FUNCTION_BLOCK Valvula_Saida_Digital (* Composite Function Block Type *)
  (* Standard: 61499-2 *)
  (* Version 0.0, 1/26/2026, Schneider Electric, template *)
  PACKAGE Hidryco.HidrycoLib;
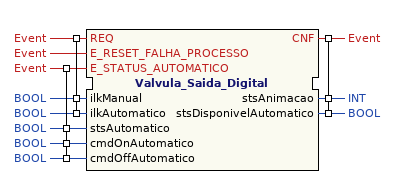
  EVENT_INPUT
    REQ WITH ilkManual, ilkAutomatico; (* Normal Execution Request *)
    E_RESET_FALHA_PROCESSO;
    E_STATUS_AUTOMATICO WITH cmdOnAutomatico, cmdOffAutomatico, stsAutomatico;
  END_EVENT
  EVENT_OUTPUT
    CNF WITH stsAnimacao, stsDisponivelAutomatico;
  END_EVENT
  VAR_INPUT
    ilkManual : BOOL;
    ilkAutomatico : BOOL;
    stsAutomatico : BOOL;
    cmdOnAutomatico : BOOL;
    cmdOffAutomatico : BOOL;
  END_VAR
  VAR_OUTPUT
    stsAnimacao : INT;
    stsDisponivelAutomatico : BOOL;
  END_VAR
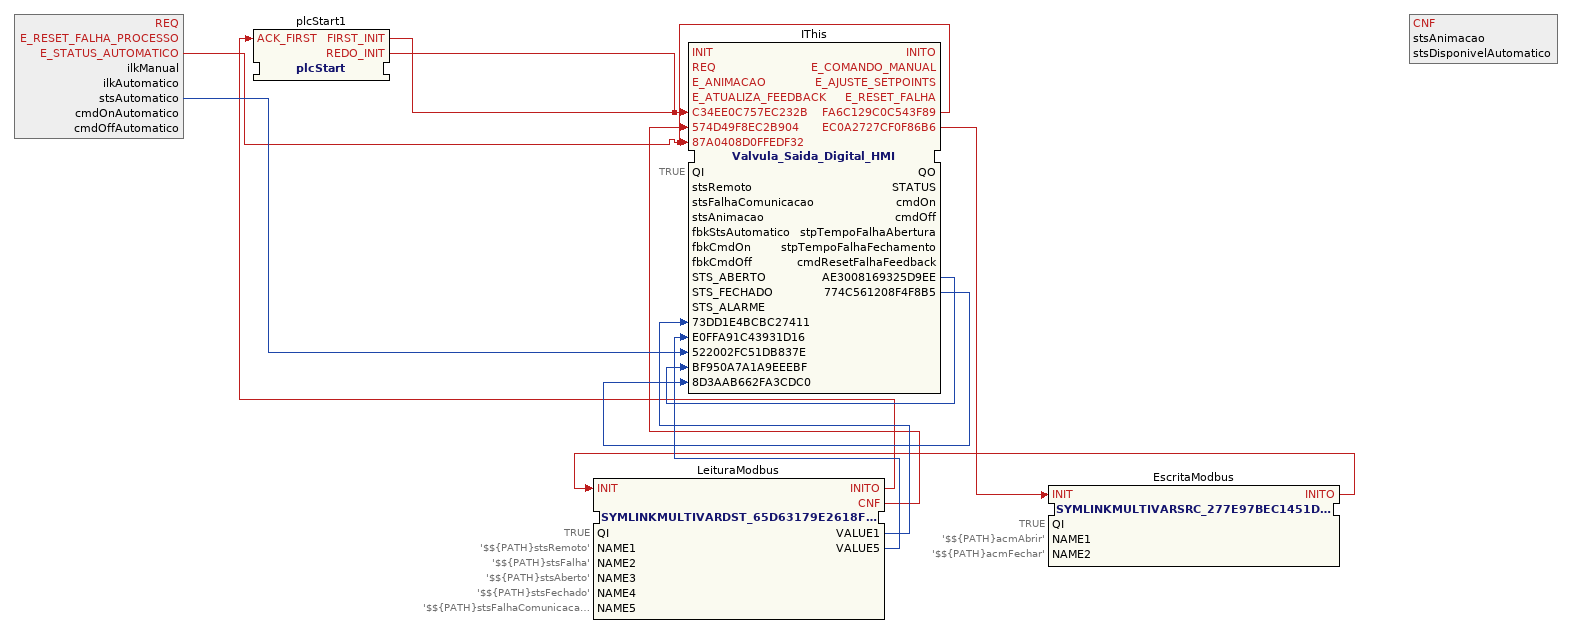
  FBS
    IThis : Valvula_Saida_Digital_HMI(QI := TRUE);
    LeituraModbus : SYMLINKMULTIVARDST_65D63179E2618F5E(QI := TRUE, NAME1 := '$${PATH}stsRemoto', NAME2 := '$${PATH}stsFalha', NAME3 := '$${PATH}stsAberto', NAME4 := '$${PATH}stsFechado', NAME5 := '$${PATH}stsFalhaComunicacao'); {SET_ATTRIBUTE(Configuration.GenericFBType.InterfaceParams, Runtime.System#I:=5;VALUE${I$}:BOOL,BOOL,BOOL,BOOL,BOOL)}
    plcStart1 : plcStart;
    EscritaModbus : SYMLINKMULTIVARSRC_277E97BEC1451D2C(QI := TRUE, NAME1 := '$${PATH}acmAbrir', NAME2 := '$${PATH}acmFechar'); {SET_ATTRIBUTE(Configuration.GenericFBType.InterfaceParams, Runtime.System#I:=2;VALUE${I$}:BOOL,BOOL)}
  END_FBS
  EVENT_CONNECTIONS
    EscritaModbus.INITO TO LeituraModbus.INIT;
    LeituraModbus.INITO TO plcStart1.ACK_FIRST;
    plcStart1.FIRST_INIT TO IThis.C34EE0C757EC232B;
    plcStart1.REDO_INIT TO IThis.C34EE0C757EC232B;
    LeituraModbus.CNF TO IThis.574D49F8EC2B904;
    IThis.FA6C129C0C543F89 TO IThis.87A0408D0FFEDF32;
    E_STATUS_AUTOMATICO TO IThis.87A0408D0FFEDF32;
    IThis.EC0A2727CF0F86B6 TO EscritaModbus.INIT;
  END_CONNECTIONS
  DATA_CONNECTIONS
    LeituraModbus.VALUE1 TO IThis.73DD1E4BCBC27411;
    LeituraModbus.VALUE5 TO IThis.E0FFA91C43931D16;
    stsAutomatico TO IThis.522002FC51DB837E;
    IThis.AE3008169325D9EE TO IThis.BF950A7A1A9EEEBF;
    IThis.774C561208F4F8B5 TO IThis.8D3AAB662FA3CDC0;
  END_CONNECTIONS
END_FUNCTION_BLOCK
